// TwinCAT 3 PLC project TcToolkitSample
// ProjectVersion: 3.1.4024.12
// project tree:
//   DUTs/ E_StationState.TcDUT (not stored), E_Command.TcDUT (not stored), ST_Status.TcDUT, ST_StationStatus.TcDUT (not stored), ST_Recipe.TcDUT, U_Word.TcDUT (not stored), T_Ident.TcDUT (not stored)
//   GVLs/ GVL_Io.TcGVL, GVL_System.TcGVL (not stored), GVL_Hmi.TcGVL (not stored)
//   POUs/Interfaces/ I_Resettable.TcIO, I_Diagnosable.TcIO (not stored), I_Station.TcIO
//   POUs/Actuators/ FB_Cylinder.TcPOU (not stored)
//   POUs/Machine/ FB_Station.TcPOU, FB_StationDerived.TcPOU
//   POUs/ MAIN.TcPOU (not stored), P_Startup.TcPOU (not stored), F_Scale.TcPOU (not stored)

// ---- DUTs/ST_Status.TcDUT
TYPE ST_Status :
STRUCT
	bBusy, bDone, bError	: BOOL;
	nErrorId			: UDINT;
END_STRUCT
END_TYPE

// ---- DUTs/ST_Recipe.TcDUT
TYPE ST_Recipe :
STRUCT
	aSteps	: ARRAY[1..8] OF INT;
	fSpeed	: LREAL;
	sId		: STRING(15);
END_STRUCT
END_TYPE

// ---- GVLs/GVL_Io.TcGVL
{attribute 'qualified_only'}
VAR_GLOBAL
	bExtendOut, bRetractOut, bSensorExtended, bSensorRetracted : BOOL;
END_VAR

// ---- POUs/Interfaces/I_Resettable.TcIO
INTERFACE I_Resettable

METHOD Reset : BOOL
END_METHOD

END_INTERFACE

// ---- POUs/Interfaces/I_Station.TcIO
INTERFACE I_Station EXTENDS I_Resettable, I_Diagnosable

METHOD Execute : BOOL
END_METHOD

PROPERTY State : E_StationState
GET
END_GET
END_PROPERTY

END_INTERFACE

// ---- POUs/Machine/FB_Station.TcPOU
FUNCTION_BLOCK FB_Station IMPLEMENTS I_Station
VAR
	refCylinder	: REFERENCE TO FB_Cylinder;
	_eState		: E_StationState;
	_eCommand	: E_Command;
	_stStatus	: ST_StationStatus;
	_stRecipe	: ST_Recipe;
	_uWord		: U_Word;
	_sIdent		: T_Ident;
	_nErrorId	: UDINT;
END_VAR

Cyclic();

METHOD Cyclic
VAR
	bExtended	: BOOL;
END_VAR
bExtended := refCylinder.bIsExtended;

CASE _eState OF
	E_StationState.Idle:
		IF _eCommand = E_Command.Start THEN
			_eState := E_StationState.Running;
		END_IF

	E_StationState.Running:
		IF bExtended THEN
			refCylinder.Retract();
		ELSE
			refCylinder.Extend();
		END_IF
		IF _nErrorId <> 0 THEN
			_eState := E_StationState.Error;
		END_IF

	E_StationState.Error:
		_stStatus.bError := TRUE;

	E_StationState.Done:
		_stStatus.bDone := TRUE;
END_CASE

_stStatus.eState := _eState;
_stStatus.nErrorId := _nErrorId;
_uWord.nWord := _stRecipe.aSteps[1];
END_METHOD

METHOD Execute : BOOL
VAR
END_VAR
IF _eState = E_StationState.Idle THEN
	_eCommand := E_Command.Start;
	_stStatus.bBusy := TRUE;
	Execute := TRUE;
ELSE
	Execute := FALSE;
END_IF
END_METHOD

METHOD Reset : BOOL
VAR
END_VAR
_eState := E_StationState.Idle;
_eCommand := E_Command.None;
_nErrorId := 0;
_stStatus.bBusy := FALSE;
_stStatus.bDone := FALSE;
_stStatus.bError := FALSE;
_stStatus.nErrorId := 0;
Reset := TRUE;
END_METHOD

PROPERTY State : E_StationState
GET
State := _eState;
END_GET
SET
_eState := State;
END_SET
END_PROPERTY

PROPERTY ErrorId : UDINT
GET
ErrorId := _nErrorId;
END_GET
END_PROPERTY

ACTION Act_Home:
refCylinder REF= GVL_System.fbCylinder;
refCylinder.Retract();
_eState := E_StationState.Idle;
_sIdent := 'STATION-01';
END_ACTION

END_FUNCTION_BLOCK

// ---- POUs/Machine/FB_StationDerived.TcPOU
FUNCTION_BLOCK FB_StationDerived EXTENDS FB_Station
VAR
	_nCycles	: UDINT;
END_VAR

Cyclic();

METHOD Cyclic
VAR
END_VAR
SUPER^.Cyclic();
_nCycles := _nCycles + 1;
END_METHOD

END_FUNCTION_BLOCK
